{attribute 'qualified_only'}
{attribute 'strict'}
TYPE E_Gripper :
(
	enum_member := 0
);
END_TYPE

(* stored: Version 1.1.0.1, ProductVersion 3.1.4024.12
   DUT E_Gripper: Id {8cadf88d-297a-4955-bc9d-05a4c1917433} *)
